TYPE ST_EPSLimits :
STRUCT
    {attribute 'pytmc' := '
        pv: FwdLimit
        io: io
    '}
    fFwd_Limits : REAL;
    {attribute 'pytmc' := '
        pv: BwdLimit
        io: io
    '}
    fBwd_Limits	: REAL;
    {attribute 'pytmc' := 'pv: ST'}
    stEPS 		: DUT_EPS;
END_STRUCT
END_TYPE

(* stored: Version 1.1.0.1, ProductVersion 3.1.4024.12
   DUT ST_EPSLimits: Id {4ee57205-73a9-412c-b8d8-c1dfce7e0790} *)
